TYPE Block128Words :
UNION
	reserved : ARRAY[1..128] OF WORD;
	unit : commUnitGeneric;
	material : materialBlock;
END_UNION
END_TYPE

(* stored: Version 1.1.0.1, ProductVersion 3.1.4022.10
   DUT Block128Words: Id {a1c10429-ec0f-4897-b3be-6badeb08a65f} *)
